// TIA Portal V15 export
// export: Created 2019-02-11T17:35:19.3274613Z, ExportSetting WithDefaults, WithReadOnly, DisplayName Totally Integrated Automation Portal, DisplayVersion V15 Update 2, DisplayName TIA Portal Openness, DisplayVersion V15 Update 2, DisplayName STEP 7 Professional, DisplayVersion V15 Update 2, DisplayName STEP 7 Safety, DisplayVersion V15, DisplayName WinCC Professional, DisplayVersion V15 Update 2, DisplayName SIMATIC Visualization Architect, DisplayVersion V15 Update 1
DATA_BLOCK "FGDB_ROBNAME@Gluing"   // DB9
{ S7_Optimized_Access := 'FALSE' }
AUTHOR : integra
FAMILY : SUB
VERSION : 1.0
// stored: AutoNumber true, CodeModifiedDate 2019-02-11T17:31:18.3581736Z, CompileDate 2019-02-11T17:35:11.3010559Z, CreationDate 2019-02-11T17:31:18.2724887Z, DBAccessibleFromOPCUA true, InstanceOfName iSF_TECH_ROBOT_GLUEING, InstanceOfNumber 19, InstanceOfType FB, InterfaceModifiedDate 2018-12-19T14:42:05.8410932Z, IsConsistent true, IsKnowHowProtected false, ModifiedDate 2019-02-11T17:31:18.3581736Z, ParameterModified 2018-06-04T13:00:21.7462385Z, StructureModified 2018-08-10T07:05:57.5964861Z, UDAEnableTagReadback false
"iSF_TECH_ROBOT_GLUEING"
   // VAR_INPUT
   //    fct : Int;
   //    safetyStop : Bool;
   //    resetResult : Bool;
   //    requestPurge2C : Bool;
   //    resetHeatting : Bool;
   //    energySaving : Bool;
   // END_VAR
   // VAR_OUTPUT
   //    applicationNOK : Bool;
   //    purgingAcitv : Bool;
   //    purgingRequest : Bool;
   //    baseInMixer2C : Bool;
   //    fault : Bool;
   // END_VAR
   // VAR_IN_OUT
   //    IfcFGExternal : "iUDT_IFC_SYS_EXTERNAL_ALARM";
   //    IfcTECH : "iUDT_IFC_ROBOT_TECH";
   //    In_PI_TECH : "iUDT_PI_ROBOT_ADRxx48_TECH";
   //    OUT_PO_TECH : "iUDT_PO_ROBOT_ADRxx48_TECH";
   // END_VAR
   // VAR
   //    F : Struct
   //       wrongID : Bool;
   //       oNoAppErrEx : Bool;
   //       oNoSysErrEx : Bool;
   //    END_STRUCT;
   //    W : Struct
   //       oDosAutoEx : Bool;
   //       oSimuOnEx : Bool;
   //       oLubricationOKEx : Bool;
   //       oBarrelNearEmtyEx : Bool;
   //       o2K_1kPurgeContFullEx : Bool;
   //       o2K_2kPurgeContFullEx : Bool;
   //       advWarning : Bool;
   //    END_STRUCT;
   //    Masks : Struct
   //       disableFault1_8 : Byte;
   //       prodRelevantFault1_8 : Byte;
   //       prodRelevantWarningt_1_8 : Byte;
   //    END_STRUCT;
   //    LastState : Struct
   //       fault1_8 : Byte;
   //       warning_1_8 : Byte;
   //    END_STRUCT;
   //    Tmr : Struct
   //       s1 { S7_SetPoint := 'True'} : Int;
   //       a1 : Int;
   //    END_STRUCT;
   //    VCB : Struct
   //       bHTReset : Bool;
   //       bEnSavEx : Bool;
   //    END_STRUCT;
   //    TmrB : Struct
   //       "1_EnableDelayTime" : Bool;
   //       "1_RunDelayTime" : Bool;
   //       "1_DoneDelayTime" : Bool;
   //    END_STRUCT;
   //    D : Struct
   //       bEnSavEx : Bool;
   //       resetResult : Bool;
   //       applicationNOK : Bool;
   //    END_STRUCT;
   //    TECH_IN : Struct
   //       ID : Byte;
   //       oReadyEx : Bool;
   //       oNoAppErrEx : Bool;
   //       oNoSysErrEx : Bool;
   //       oDosAutoEx : Bool;
   //       oSimuOnEx : Bool;
   //       oMeasurActivEx : Bool;
   //       oLubricationOKEx : Bool;
   //       oBarrelNearEmtyEx : Bool;
   //       oHeatingOnEx : Bool;
   //       oHeatingIOEx : Bool;
   //       oPumpIOEx : Bool;
   //       oPurgingActivEx : Bool;
   //       oLiveBitEx : Bool;
   //       o2K_PrewarningPottimeEx : Bool;
   //       oEnergyModeOnEx : Bool;
   //       o2K_Base_1K_in_MixerEx : Bool;
   //       o2K_1kPurgeContFullEx : Bool;
   //       o2K_2kPurgeContFullEx : Bool;
   //       oReqPurgingEx : Bool;
   //       STOactive : Bool;
   //       advWarning : Bool;
   //       technoBit22 : Bool;
   //       technoBit23 : Bool;
   //       technoBit24 : Bool;
   //       technoBit25 : Bool;
   //       technoBit26 : Bool;
   //       technoBit27 : Bool;
   //       technoBit28 : Bool;
   //       technoBit29 : Bool;
   //       technoBit30 : Bool;
   //       technoBit31 : Bool;
   //       technoBit32 : Bool;
   //       technoBit33 : Bool;
   //       technoBit34 : Bool;
   //       technoBit35 : Bool;
   //       technoBit36 : Bool;
   //       technoBit37 : Bool;
   //       technoBit38 : Bool;
   //       technoBit39 : Bool;
   //       technoBit40 : Bool;
   //    END_STRUCT;
   //    TECH_OUT : Struct
   //       ID : Byte;
   //       bQuittEx : Bool;
   //       bSysOnEx : Bool;
   //       bEnSavEx : Bool;
   //       b2KpurgBa : Bool;
   //       bOperRele : Bool;
   //       bHTReset : Bool;
   //       resetResult : Bool;
   //       technoBit8 : Bool;
   //       technoBit9 : Bool;
   //       technoBit10 : Bool;
   //       technoBit11 : Bool;
   //       technoBit12 : Bool;
   //       technoBit13 : Bool;
   //       technoBit14 : Bool;
   //       technoBit15 : Bool;
   //       technoBit16 : Bool;
   //       technoBit17 : Bool;
   //       technoBit18 : Bool;
   //       technoBit19 : Bool;
   //       technoBit20 : Bool;
   //       technoBit21 : Bool;
   //       technoBit22 : Bool;
   //       technoBit23 : Bool;
   //       technoBit24 : Bool;
   //       technoBit25 : Bool;
   //       technoBit26 : Bool;
   //       technoBit27 : Bool;
   //       technoBit28 : Bool;
   //       technoBit29 : Bool;
   //       technoBit30 : Bool;
   //       technoBit31 : Bool;
   //       technoBit32 : Bool;
   //       technoBit33 : Bool;
   //       technoBit34 : Bool;
   //       technoBit35 : Bool;
   //       technoBit36 : Bool;
   //       technoBit37 : Bool;
   //       technoBit38 : Bool;
   //       technoBit39 : Bool;
   //       technoBit40 : Bool;
   //    END_STRUCT;
   //    IEC_Timer_bHTReset : TP_TIME;
   //    IEC_Timer_ack : TP_TIME;
   // END_VAR
BEGIN
END_DATA_BLOCK
